Universal Robots PolyScope program: rtde_control_loop_move_unified_only.urp

Program rtde_control_loop_move_unified_only (installation=default directory=/programs/usbdisk createdIn=3.2.19275.0 lastSavedIn=3.10.1.76190 robotSerialNumber=2015330464)
Calibrated DH parameters: a=[-0.000078, -0.24255, -0.20675, 0.000027, 0.00005, 0]; d=[0.151929, 6.023359, 2.368486, -8.27907, 0.085262, 0.082386]; alpha=[1.570912, 0.005147, 0.006417, 1.571047, -1.570606, 0]; deltaTheta=[-0.000006, 0.127022, 0.127628, -0.254788, 0.000059, -0.000009]
InitVariablesNode variables(variable(name=init_move, expression=1), variable(name=init_tsk, expression=0), variable(name=qpos, expression=[0,0,0,0,0,0]), variable(name=tsk_spc, expression=0), variable(name=xpos, expression=Base))
BeforeStart
  Script: init_tsk=read_input_integer_register(2)
  Script: tsk_spc=read_input_integer_register(1)
  Script: write_output_integer_register(0,0)
  Script: rtde_set_watchdog("input_int_register_0", 1, "PAUSE")
Robot Program (runOnlyOnce=false)
  If init_move≟1
    Script: sync()
    If init_tsk≟1
      MoveL speed 25 mm/s, acceleration 120 mm/s^2 (useActiveTCP=false) tcp=TCP_1; feature=Base
        Waypoint Waypoint (Variable): variable(name=xpos)
    Else 
      MoveJ speed 30 deg/s, acceleration 40 deg/s^2 (useActiveTCP=false)
        Waypoint Waypoint (Variable): variable(name=qpos)
    Popup Message (haltProgram=false message=Robot configuration is now at the initial state. inputType=Text)
    Wait Sleep waitTime=0.01
    Script: write_output_integer_register(0, 1)
    Script: sync()
    init_move := 0
  Else 
    If read_input_integer_register(3)≟1
      Script: servoj(qpos)
    Else 
      Script: stopj(2)
      Popup Message (haltProgram=true message=End of motion inputType=Text)
Thread Thread_1 (runOnlyOnce=false trackProgramExecution=false)
  Loop Forever
    If tsk_spc≟1
      tmp := p[0,0,0,0,0,0]
    Else 
      tmp := [0,0,0,0,0,0]
    Script: tmp[0] = read_input_float_register(0)
    Script: tmp[1] = read_input_float_register(1)
    Script: tmp[2] = read_input_float_register(2)
    Script: tmp[3] = read_input_float_register(3)
    Script: tmp[4] = read_input_float_register(4)
    Script: tmp[5] = read_input_float_register(5)
    If tsk_spc≟1
      If tmp != p[0,0,0,0,0,0]
        xpos := tmp
        qpos := get_inverse_kin(xpos)
    Else 
      If tmp != [0,0,0,0,0,0]
        qpos := tmp
        xpos := get_target_tcp_pose()
    Script: sync()
